INTERFACE I_MasterArmCtrl

METHOD reset : BOOL
VAR_INPUT
END_VAR
END_METHOD

METHOD run : BOOL
VAR_IN_OUT CONSTANT
	i_shoulderPose :ARRAY[1..2] OF ST_Frame;
	i_slaveStatus :ST_SlaveStatus;
END_VAR
VAR_IN_OUT
	i_masterArms :ARRAY[1..g_mArmNum] OF FB_MasterArm;
END_VAR
END_METHOD

END_INTERFACE

(* stored: Version 1.1.0.1, ProductVersion 3.1.4024.12
   Itf I_MasterArmCtrl: Id {f0c76191-353c-4edd-a51a-aab3c6b7f25c}
   Method reset: Id {d3d01b04-dfab-450f-8fd4-a152b95c8241}
   Method run: Id {cdc1ac69-5bc1-4174-b158-da097af4b3d6} *)
